FUNCTION_BLOCK PLUNGE_TOOLAXIS_STRATEGY
  (* Standard: 61499-2 *)
  (* Version 1.0, 17-05-12, GASR, Universidade do Estado de Santa Catarina *)
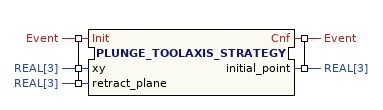
  EVENT_INPUT
    Init WITH xy, retract_plane;
  END_EVENT
  EVENT_OUTPUT
    Cnf WITH initial_point;
  END_EVENT
  VAR_INPUT
    xy : ARRAY [0..2] OF REAL;
    retract_plane : ARRAY [0..2] OF REAL;
  END_VAR
  VAR_OUTPUT
    initial_point : ARRAY [0..2] OF REAL;
  END_VAR
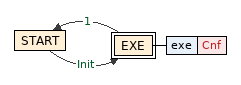
  EC_STATES
    EXE : exe -> Cnf;
    START;
  END_STATES
  EC_TRANSITIONS
    START TO EXE := Init;
    EXE TO START := 1;
  END_TRANSITIONS
  ALGORITHM exe IN Lua:
 initial_point[1] = xy[1] initial_point[2] = xy[2] initial_point[3] = retract_plane[3]
  END_ALGORITHM
END_FUNCTION_BLOCK
